// TIA Portal project "ISA_P4a" (V16)

(* hardware
DEVICE "S7-1200 station_1"  S7-1200 Station
   slot 0: "Rack_0"  S7-1200 Rack  Rack  V1.0
   slot 1: "PLC_1"  CPU 1215C DC/DC/DC  6ES7 215-1AG40-0XB0  V4.4
DEVICE "PC-System_1"  SIMATIC PC station
   slot 0: "Estación PC SIMATIC"  Rail  SIMATIC PC-Station  V1.0
      slot 125: "Stationmanager"  Station_Manager  V6.0.4
   slot 1: "HMI_RT_1"  WinCC RT Advanced  6AV2 104-0xxxx-xxxx  16.0.0.0
      slot 33792: "Interfaz del equipo"  Host interface
   slot 2: "IE general_1"  IE General  IE_CP  V8.2.0
*)

// ===== PLC "PLC_1"  CPU 1215C DC/DC/DC =====

VAR_GLOBAL   // PLC tag table "Tabla de variables estándar"
   "Tag_1" AT %Q0.0 : Bool;
   "Encoder" AT %ID1000 : DWord;
   "Sync" AT %I0.3 : Bool;
   "Gate" AT %I1.0 : Bool;
END_VAR

DATA_BLOCK "Variables"   // DB1
{ S7_Optimized_Access := 'TRUE' }
VERSION : 0.1
   VAR
      resolution : Int;
      diameter : Int;
      distance : Int;
   END_VAR
BEGIN
END_DATA_BLOCK

ORGANIZATION_BLOCK "Main"   // OB1, LAD, ProgramCycle
TITLE = "Main Program Sweep (Cycle)"
{ S7_Optimized_Access := 'TRUE' }
VERSION : 0.1
   VAR_INPUT
      Initial_Call : Bool;   // Initial call of this OB
      Remanence : Bool;   // =True, if remanent data are available
   END_VAR
BEGIN
END_ORGANIZATION_BLOCK

ORGANIZATION_BLOCK "Hardware interrupt"   // OB40, LAD, HWProcessInterrupt
{ S7_Optimized_Access := 'TRUE' }
VERSION : 0.1
   VAR_INPUT
      LADDR : Hw_Io;   // Hardware identifier
      USI : Word;   // User structure identifier
      IChannel : USInt;   // Interrupt channel number
      EventType : Byte;   // EventType
   END_VAR
BEGIN

REGION Network 1
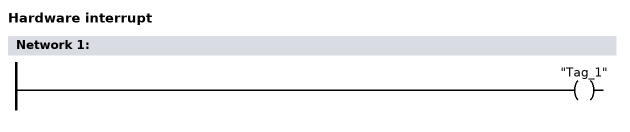
   RUNG wire#powerrail
      Coil( "Tag_1" )
   END_RUNG
   // the same network as SCL:
   "Tag_1" := TRUE;
END_REGION
END_ORGANIZATION_BLOCK

ORGANIZATION_BLOCK "Cálculos"   // OB123, LAD, ProgramCycle
TITLE = "Main Program Sweep (Cycle)"
{ S7_Optimized_Access := 'TRUE' }
VERSION : 0.1
   VAR_INPUT
      Initial_Call : Bool;   // Initial call of this OB
      Remanence : Bool;   // =True, if remanent data are available
   END_VAR
   VAR CONSTANT
      pi : Real := 3.14169;
   END_VAR
BEGIN

REGION Network 1 (SCL)
   "Variables".distance := ("Encoder" * "Variables".diameter * #pi) / "Variables".resolution;
END_REGION
END_ORGANIZATION_BLOCK

(* ===== HMI "HMI_RT_1" =====
system functions are stored by id; their names below are inferred from use
connection "HMI_Conexión_1": ETHERNET, S7_1200_OMS

HMI tags "Tabla de variables estándar"
   "Variables_distance" : Int = PLC Variables.distance, 1 s
   "Variables_Resolution" : Int = PLC Variables.resolution, 1 s
   "Variables_Diámeter" : Int = PLC Variables.diameter, 1 s
   "Tag_1" : Bool = PLC Tag_1 AT %Q0.0, 1 s
   "Encoder" : DWord = PLC Encoder AT %ID1000, 1 s

screen "Imagen_1" 800x600
   IOField "Campo ES_1" at 342,237 size 96x32; FormatPattern s99999
      ProcessValue <- "Variables_distance"
   IOField "Campo ES_2" at 164,143 size 96x32; FormatPattern 99999
      ProcessValue <- "Variables_Resolution"
   IOField "Campo ES_3" at 519,143 size 96x32; FormatPattern 99999
      ProcessValue <- "Variables_Diámeter"
   TextField "Campo de texto_1" at 290,206 size 196x22; Text 'distancia recorrida (mm):'
   TextField "Campo de texto_2" at 148,108 size 130x22; Text 'Resolución (ppr)'
   TextField "Campo de texto_3" at 508,108 size 118x22; Text 'Diámetro (mm)'
   Button "Botón_1" at 341,447 size 96x32; TextOff 'off'
      on Press: ResetBit("Tag_1")
   TextField "Campo de texto_4" at 360,317 size 58x22; Text 'pulsos:'
   IOField "Campo ES_4" at 323,350 size 143x32; FormatPattern 9999999999
      ProcessValue <- "Encoder"
*)